(* PLC project Generated.project, CODESYS CODESYS V3.5 SP19 Patch 1 *)
(* stored: creationDateTime 2026-08-31T12:26:56.544484, modificationDateTime 2026-08-31T12:26:56.544484 *)

(* values of E_DiveSearchState: WAIT_PRECONDITIONS: Attente benne ouverte, positions et Kobold au repos; READY_TO_DESCEND: Prêt à assister une demande de descente; SEARCHING_IMMERSION: Descending : attente front 0->1 dans fenêtre eau; SEARCHING_BOTTOM: Immersion validée : attente front 1->0 au fond; BOTTOM_CONFIRMED: Fond validé ; extraction peut être demandée; ERROR_HOLD: Séquence invalide, descente assistée interdite *)

{attribute 'qualified_only'}
{attribute 'strict'}
TYPE E_DiveSearchState : (WAIT_PRECONDITIONS := 0, READY_TO_DESCEND := 1, SEARCHING_IMMERSION := 2, SEARCHING_BOTTOM := 3, BOTTOM_CONFIRMED := 4, ERROR_HOLD := 5);
END_TYPE

(* ======================================================================= 🧩 ST_Fault — Brique socle défaut (2 vues : live + latchée) ─────────────────────────────────────────────────────────────── 🎯 Rôle : porter l'état défaut d'un composant, applicable dans TOUS les cas (acquittable ou non), sans brique warning séparée. • Vue LIVE (Error / ErrorId) : suit la cause, retombe seule à 0. • Vue LATCHÉE (Latched / LatchedId): mémorisée au défaut, reste jusqu'au front Reset. Le choix acquittable / non-acquittable se fait PAR CAUSE (ST_FaultCause.Latching), jamais par bloc. 🔒 Sécurité : interlock TOUJOURS sur la cause brute (Error / ErrorId), jamais sur l'acquittement. Reset TOUJOURS effectif, jamais conditionné (std §9). 🧬 Composition : brique de base réutilisable — sortie de FB, struct métier, GVL. Texte IHM NON stocké ici : dérivé côté IHM depuis LatchedId / ErrorId. 📄 Doc : DOC/STDS/CODE_QUALITY_STANDARDS.md §2quinquies / §9 ======================================================================= *)
TYPE ST_Fault : STRUCT
  Error : BOOL;  (* <-- [DIAG] vue LIVE : au moins une cause présente maintenant *)
  ErrorId : WORD;  (* <-- [DIAG] bitfield des causes présentes maintenant (0 si aucune) *)
  Latched : BOOL;  (* <-- [DIAG] vue LATCHÉE : défaut non acquitté, reste jusqu'au front Reset *)
  LatchedId : WORD;  (* <-- [DIAG] ErrorId figé à l'apparition du défaut, effacé au Reset *)
END_STRUCT;
END_TYPE

(* ======================================================================= 🧩 ST_FaultCause — Cause élémentaire alimentant ST_Fault (socle FB_FaultCore) ─────────────────────────────────────────────────────────────── 🎯 Rôle : une cause exprimée EN CLAIR (BOOL + libellé), sans bitfield ni masque. Le FB métier remplit une liste (ARRAY[0..15] OF ST_FaultCause) ; le socle FB_FaultCore en déduit ST_Fault (vue live + vue latchée). 🔒 Sécurité : interlock TOUJOURS sur Active (cause brute), jamais sur le latch. Latching = TRUE → la cause ARME la vue latchée (défaut à acquitter). Latching = FALSE → la cause n'alimente que la vue live (retombe seule). Fail-safe : une cause laissée à Latching=FALSE reste visible en live — pour la rendre acquittable, il faut le déclarer explicitement. 📄 Doc : DOC/STDS/CODE_QUALITY_STANDARDS.md §2quinquies / §9 ======================================================================= *)
TYPE ST_FaultCause : STRUCT
  Active : BOOL;  (* 1 = cause présente maintenant (interlock sur cette valeur) *)
  Latching : BOOL;  (* 1 = cause à acquitter (arme Latched) ; 0 = live seulement *)
  Texte : STRING;  (* libellé prêt IHM (non stocké dans ST_Fault, dérivé côté IHM) *)
END_STRUCT;
END_TYPE

(* ======================================================================= 🧩 ST_Lifecycle — Brique socle cycle d'exécution ─────────────────────────────────────────────────────────────── 🎯 Rôle : porter l'avancement d'une action à cycle (organe, séquenceur). Optionnelle : un FB purement synchrone (conditionneur, filtre, joystick) ne la porte pas. 🧬 Composition : brique de base réutilisable, composée avec ST_Fault. 📄 Doc : DOC/STDS/CODE_QUALITY_STANDARDS.md §2quinquies ======================================================================= *)
TYPE ST_Lifecycle : STRUCT
  Busy : BOOL;  (* <-- [STAT] 1 = action en cours *)
  Done : BOOL;  (* <-- [STAT] 1 = action terminée avec succès *)
END_STRUCT;
END_TYPE

(* ======================================================================= ST_fbDiveSearch_Inputs - Bus d'entree du cycle FB_DiveSearch ======================================================================= *)
TYPE ST_fbDiveSearch_Inputs : STRUCT
  PowerContactorEngaged : BOOL;  (* === AUTORISATIONS & COMMANDE === Chaine de puissance engagee *)
  Mode : E_Mode;  (* Mode arbitre courant *)
  MotionRequestActive : BOOL;  (* Demande de mouvement couplee *)
  MotionDirection : INT;  (* Sens demande (-1 = descente) *)
  BucketIsOpen : BOOL;  (* === CAPTEURS & MESURES === Benne ouverte confirmee *)
  KoboldImmersed : BOOL;  (* Kobold immerge *)
  M1Position_M : REAL;  (* Position cable M1 (m) *)
  M2Position_M : REAL;  (* Position cable M2 (m) *)
  PositionsValid : BOOL;  (* Mesures M1/M2 valides *)
  CurrentSpeedStep : INT;  (* Palier reel courant (0..5) *)
  DiveStartMin_M : REAL;  (* === REGLAGES METIER === Position minimale avant descente (m) *)
  ImmersionUpper_M : REAL;  (* Borne haute fenetre immersion (m) *)
  ImmersionLower_M : REAL;  (* Borne basse fenetre immersion (m) *)
  CableLimitAscent_M : REAL;  (* Limite haute exploitation (m) *)
  LimitLegalDepthMin_M : REAL;  (* Limite basse legale (m) *)
  CfgDiveFloorStep : INT;  (* Plancher palier descente (0..5) *)
  CycleTime : TIME;  (* Periode d'execution du cycle *)
  BypassPreconditions : BOOL;  (* Bypass reserve au mode maintenance N2/test *)
  Config : ST_fbDiveSearch_Config;  (* Parametres timeout *)
END_STRUCT;
END_TYPE

(* ======================================================================= ST_fbDiveSearch_Outputs - Bus de sortie du cycle FB_DiveSearch ======================================================================= *)
TYPE ST_fbDiveSearch_Outputs : STRUCT
  StepState : E_DiveSearchState;  (* === ETAT DU CYCLE === Etape courante *)
  StepAtFault : E_DiveSearchState;  (* Etape figee au defaut *)
  DescendPermit : BOOL;  (* === PERMIS & ORDRES ASSISTES === Autorisation de descente assistee *)
  KoboldContactorCmd : BOOL;  (* Commande alimentation Kobold (fail-safe, coupe au front de fond) *)
  BottomTouchConfirmed : BOOL;  (* Fond confirme *)
  MinStepDown : INT;  (* Plancher palier descente *)
  OperatorActionId : WORD;  (* === DIAGNOSTIC OPERATEUR === Identifiant numerique de l'action *)
  OperatorAction : STRING(120);  (* Consigne operateur ASCII *)
END_STRUCT;
END_TYPE

(* values of E_Mode: DISABLE: Mode Désactivé / Veille de sécurité (sorties bloquées); MAINT_N1: Manuel Niveau 1 : Pilotage unitaire avec toutes sécurités actives; MAINT_N2: Manuel Niveau 2 : Pilotage dégradé (droits étendus + bypasses autorisés); SEMI_AUTO: Mode Semi-Automatique (séquenceur automatique) *)

{attribute 'qualified_only'}
{attribute 'strict'}
TYPE E_Mode : (DISABLE := 0, MAINT_N1 := 1, MAINT_N2 := 2, SEMI_AUTO := 3);
END_TYPE

(* ======================================================================= ST_fbDiveSearch_Config - Reglages du cycle de recherche du fond ======================================================================= *)
TYPE ST_fbDiveSearch_Config : STRUCT
  DiveSpeedMin_Mps : REAL := 0.15;  (* Vitesse minimale de calcul du timeout (m/s) *)
  TimeoutMarginFactor : REAL := 1.5;  (* Marge appliquee au temps theorique *)
  TimeoutMinCourse_M : REAL := 1;  (* Course minimale prise en compte (m) *)
  TimeoutMaxCourse_M : REAL := 200;  (* Course maximale prise en compte (m) *)
  SecToMs : REAL := 1000;  (* Conversion secondes vers millisecondes *)
END_STRUCT;
END_TYPE

(* ======================================================================= FB_DiveSearch - Assistance plongee et recherche du fond Kobold Role : qualifier l'immersion et autoriser la descente assistee. Interface : contrat standard + bus Inputs/Outputs. Documentation : DOC/AF/AF_Partie-04_Mode_SemiAuto_Sequenceur_v2.3.md ======================================================================= *)
FUNCTION_BLOCK FB_DiveSearch
  VAR_INPUT
    Enable : BOOL;  (* === CONTRAT STANDARD === --> [CMD] Autorisation generale du FB *)
    Reset : BOOL;  (* --> [CMD] Acquittement defaut sur front *)
    Inputs : ST_fbDiveSearch_Inputs;  (* === BUS FONCTIONNEL === --> [BUS] Commande, capteurs et reglages *)
  END_VAR
  VAR_OUTPUT
    Ready : BOOL;  (* === STATUT IEC === <-- [STAT] FB pret a fonctionner *)
    Fault : ST_Fault;  (* <-- [DIAG] Defaut live et latche *)
    Lifecycle : ST_Lifecycle;  (* <-- [STAT] Cycle en cours / termine *)
    Outputs : ST_fbDiveSearch_Outputs;  (* === BUS FONCTIONNEL === <-- [BUS] Etat, permis et diagnostic *)
  END_VAR
  VAR
    ResetEdge : R_TRIG;  (* === SOUS-INSTANCES & FRONTS === . [LOC] Front Reset *)
    ErrorEdge : R_TRIG;  (* . [LOC] Apparition d'un defaut *)
    KoboldRiseEdge : R_TRIG;  (* . [LOC] Entree dans l'eau *)
    KoboldFallEdge : F_TRIG;  (* . [LOC] Sortie de l'eau / fond *)
    instFault : FB_FaultCore;  (* * [INST] Socle defaut transverse *)
    instCauses : ARRAY[0..15] OF ST_FaultCause;  (* . [LOC] Causes nommees *)
    ImmersionCourse_M : REAL;  (* === CALCULS DE GARDE === . [LOC] Course maximale vers immersion (m) *)
    BottomCourse_M : REAL;  (* . [LOC] Course maximale vers fond (m) *)
    CalculatedImmersionTimeout : TIME;  (* . [LOC] Timeout immersion calcule *)
    CalculatedBottomTimeout : TIME;  (* . [LOC] Timeout fond calcule *)
    EffectiveDiveSpeedMin_Mps : REAL;  (* . [LOC] Vitesse minimale appliquee (m/s) *)
    EffectiveTimeoutMargin : REAL;  (* . [LOC] Marge appliquee au calcul *)
    EffectiveTimeoutMinCourse_M : REAL;  (* . [LOC] Plancher de course applique (m) *)
    EffectiveTimeoutMaxCourse_M : REAL;  (* . [LOC] Plafond de course applique (m) *)
    EffectiveSecToMs : REAL;  (* . [LOC] Conversion secondes/millisecondes *)
    ImmersionTimerAcc : TIME := TIME#0ms;  (* === MEMORISATIONS & TEMPORISATIONS === . [LOC] Temps effectif de recherche immersion *)
    BottomTimerAcc : TIME := TIME#0ms;  (* . [LOC] Temps effectif de recherche fond *)
    PrevState : E_DiveSearchState;  (* . [LOC] Etat du scan precedent *)
    ImmersionConfirmed : BOOL;  (* . [LOC] Immersion validee *)
    StepAtFaultCaptured : BOOL;  (* . [LOC] Etape de defaut deja figee *)
    ErrorCausePresent : BOOL;  (* === CAUSES INTERNES === . [LOC] Parametrage invalide *)
    SeqErrorFault : BOOL;  (* . [LOC] Incoherence de sequence *)
    Palier5ForbiddenFault : BOOL;  (* . [LOC] Palier 5 interdit sous Kobold *)
    TimeoutImmersionFault : BOOL;  (* . [LOC] Timeout recherche immersion *)
    TimeoutBottomFault : BOOL;  (* . [LOC] Timeout recherche fond *)
    DescentActive : BOOL;  (* . [LOC] Descending demandee et autorisee *)
  END_VAR

            

{region "§1 Fronts, calculs et causes"}
ResetEdge(CLK := Reset);
KoboldRiseEdge(CLK := Inputs.KoboldImmersed);
KoboldFallEdge(CLK := Inputs.KoboldImmersed);

// Les valeurs par defaut du DUT couvrent l'appel sans configuration explicite.
// Le repli runtime protege aussi un appel avec une structure entierement nulle.
EffectiveDiveSpeedMin_Mps := Inputs.Config.DiveSpeedMin_Mps;
IF EffectiveDiveSpeedMin_Mps <= 0.0 THEN EffectiveDiveSpeedMin_Mps := 0.15; END_IF;
EffectiveTimeoutMargin := Inputs.Config.TimeoutMarginFactor;
IF EffectiveTimeoutMargin <= 0.0 THEN EffectiveTimeoutMargin := 1.5; END_IF;
EffectiveTimeoutMinCourse_M := Inputs.Config.TimeoutMinCourse_M;
IF EffectiveTimeoutMinCourse_M <= 0.0 THEN EffectiveTimeoutMinCourse_M := 1.0; END_IF;
EffectiveTimeoutMaxCourse_M := Inputs.Config.TimeoutMaxCourse_M;
IF EffectiveTimeoutMaxCourse_M < EffectiveTimeoutMinCourse_M THEN EffectiveTimeoutMaxCourse_M := 200.0; END_IF;
EffectiveSecToMs := Inputs.Config.SecToMs;
IF EffectiveSecToMs <= 0.0 THEN EffectiveSecToMs := 1000.0; END_IF;

ErrorCausePresent := (Inputs.CycleTime <= T#0ms)
                 OR (NOT Inputs.BypassPreconditions AND (
                       (Inputs.DiveStartMin_M < Inputs.ImmersionUpper_M)
                    OR (Inputs.ImmersionUpper_M <= Inputs.ImmersionLower_M)
                    OR (Inputs.ImmersionLower_M <= Inputs.LimitLegalDepthMin_M)
                    OR (Inputs.CableLimitAscent_M <= Inputs.ImmersionLower_M)));

ImmersionCourse_M := LIMIT(EffectiveTimeoutMinCourse_M,
                           Inputs.CableLimitAscent_M - Inputs.ImmersionLower_M,
                           EffectiveTimeoutMaxCourse_M);
BottomCourse_M := LIMIT(EffectiveTimeoutMinCourse_M,
                        Inputs.ImmersionLower_M - Inputs.LimitLegalDepthMin_M,
                        EffectiveTimeoutMaxCourse_M);
CalculatedImmersionTimeout := UDINT_TO_TIME(REAL_TO_UDINT(
    ImmersionCourse_M / EffectiveDiveSpeedMin_Mps * EffectiveTimeoutMargin * EffectiveSecToMs));
CalculatedBottomTimeout := UDINT_TO_TIME(REAL_TO_UDINT(
    BottomCourse_M / EffectiveDiveSpeedMin_Mps * EffectiveTimeoutMargin * EffectiveSecToMs));

IF (Outputs.StepState = E_DiveSearchState.SEARCHING_IMMERSION)
   AND Inputs.MotionRequestActive AND (Inputs.MotionDirection = -1) THEN
    ImmersionTimerAcc := ImmersionTimerAcc + Inputs.CycleTime;
    IF ImmersionTimerAcc >= CalculatedImmersionTimeout THEN TimeoutImmersionFault := TRUE; END_IF;
END_IF;

IF (Outputs.StepState = E_DiveSearchState.SEARCHING_BOTTOM)
   AND Inputs.MotionRequestActive AND (Inputs.MotionDirection = -1) THEN
    BottomTimerAcc := BottomTimerAcc + Inputs.CycleTime;
    IF BottomTimerAcc >= CalculatedBottomTimeout THEN TimeoutBottomFault := TRUE; END_IF;
END_IF;

IF ResetEdge.Q AND NOT ErrorCausePresent AND NOT Inputs.KoboldImmersed
   AND NOT Inputs.MotionRequestActive AND NOT (Inputs.CurrentSpeedStep > 4) THEN
    SeqErrorFault := FALSE;
    Palier5ForbiddenFault := FALSE;
    TimeoutImmersionFault := FALSE;
    TimeoutBottomFault := FALSE;
    ImmersionTimerAcc := T#0ms;
    BottomTimerAcc := T#0ms;
    ImmersionConfirmed := FALSE;
    Outputs.BottomTouchConfirmed := FALSE;
    Outputs.StepAtFault := E_DiveSearchState.WAIT_PRECONDITIONS;
    StepAtFaultCaptured := FALSE;
    Outputs.StepState := E_DiveSearchState.WAIT_PRECONDITIONS;
END_IF;

instCauses[0].Active := SeqErrorFault;
instCauses[0].Latching := TRUE;
instCauses[0].Texte := 'Incoherence sequence immersion Kobold';
instCauses[1].Active := ErrorCausePresent;
instCauses[1].Latching := TRUE;
instCauses[1].Texte := 'Parametrage invalide des seuils de plongee';
instCauses[2].Active := Palier5ForbiddenFault;
instCauses[2].Latching := TRUE;
instCauses[2].Texte := 'Palier 5 interdit pendant la mesure Kobold';
instCauses[3].Active := TimeoutImmersionFault;
instCauses[3].Latching := TRUE;
instCauses[3].Texte := 'Timeout recherche immersion Kobold';
instCauses[4].Active := TimeoutBottomFault;
instCauses[4].Latching := TRUE;
instCauses[4].Texte := 'Timeout recherche fond Kobold';

instFault(Enable := Enable, Reset := Reset, Causes := instCauses);
Fault := instFault.Fault;

ErrorEdge(CLK := Fault.Error);
IF ErrorEdge.Q AND NOT StepAtFaultCaptured THEN
    Outputs.StepAtFault := PrevState;
    StepAtFaultCaptured := TRUE;
ELSIF ResetEdge.Q AND NOT ErrorCausePresent AND NOT Inputs.KoboldImmersed
      AND NOT Inputs.MotionRequestActive AND NOT (Inputs.CurrentSpeedStep > 4) THEN
    Outputs.StepAtFault := E_DiveSearchState.WAIT_PRECONDITIONS;
END_IF;
{endregion}

{region "§2 Neutralisation et machine d'etat"}
IF NOT Enable OR NOT Inputs.PowerContactorEngaged THEN
    Ready := FALSE;
    Lifecycle.Busy := FALSE;
    Lifecycle.Done := FALSE;
    Outputs.DescendPermit := FALSE;
    Outputs.KoboldContactorCmd := FALSE;
    Outputs.BottomTouchConfirmed := FALSE;
    Outputs.StepState := E_DiveSearchState.WAIT_PRECONDITIONS;
    Outputs.OperatorActionId := 0;
    Outputs.OperatorAction := '';
    ImmersionConfirmed := FALSE;
    ImmersionTimerAcc := T#0ms;
    BottomTimerAcc := T#0ms;
    Outputs.MinStepDown := 0;
    PrevState := E_DiveSearchState.WAIT_PRECONDITIONS;
    RETURN;
END_IF;

Ready := Enable AND NOT Fault.Latched;
Outputs.DescendPermit := FALSE;
Outputs.KoboldContactorCmd := FALSE;
Lifecycle.Busy := FALSE;
Lifecycle.Done := FALSE;
Outputs.OperatorActionId := 0;
Outputs.OperatorAction := '';

DescentActive := Inputs.MotionRequestActive AND (Inputs.MotionDirection = -1)
              AND ((Inputs.Mode = E_Mode.MAINT_N1) OR (Inputs.Mode = E_Mode.MAINT_N2))
              AND NOT (Inputs.CurrentSpeedStep > 4)
              AND NOT SeqErrorFault;

IF Fault.Error OR Fault.Latched THEN
    Outputs.StepState := E_DiveSearchState.ERROR_HOLD;
    Outputs.KoboldContactorCmd := FALSE;
    Outputs.OperatorActionId := 16#0180;
    Outputs.OperatorAction := 'Verifier les conditions puis rearmer avant une nouvelle plongee.';
ELSE
    CASE Outputs.StepState OF
        E_DiveSearchState.WAIT_PRECONDITIONS:
            IF NOT Inputs.BypassPreconditions
               AND (NOT Inputs.BucketIsOpen OR NOT Inputs.PositionsValid OR Inputs.KoboldImmersed
                    OR (Inputs.M1Position_M < Inputs.DiveStartMin_M)
                    OR (Inputs.M2Position_M < Inputs.DiveStartMin_M)) THEN
                Outputs.OperatorActionId := 16#0100;
                Outputs.OperatorAction := 'Verifier benne ouverte, positions et Kobold au repos.';
            ELSE
                Outputs.StepState := E_DiveSearchState.READY_TO_DESCEND;
            END_IF;

        E_DiveSearchState.READY_TO_DESCEND:
            Ready := TRUE;
            Outputs.OperatorActionId := 16#0101;
            Outputs.OperatorAction := 'Demander une descente pour rechercher le fond.';
            IF Inputs.MotionRequestActive AND (Inputs.MotionDirection = -1) THEN
                ImmersionTimerAcc := T#0ms;
                Outputs.StepState := E_DiveSearchState.SEARCHING_IMMERSION;
            END_IF;

        E_DiveSearchState.SEARCHING_IMMERSION:
            Lifecycle.Busy := TRUE;
            Outputs.DescendPermit := DescentActive;
            Outputs.KoboldContactorCmd := DescentActive;
            Outputs.OperatorActionId := 16#0102;
            Outputs.OperatorAction := 'Maintenir la descente : recherche immersion Kobold.';
            IF Inputs.CurrentSpeedStep > 4 THEN
                IF NOT StepAtFaultCaptured THEN
                    Outputs.StepAtFault := Outputs.StepState;
                    StepAtFaultCaptured := TRUE;
                END_IF;
                Palier5ForbiddenFault := TRUE;
            END_IF;
            IF KoboldRiseEdge.Q THEN
                IF (Inputs.M1Position_M <= Inputs.ImmersionUpper_M)
                   AND (Inputs.M1Position_M >= Inputs.ImmersionLower_M)
                   AND (Inputs.M2Position_M <= Inputs.ImmersionUpper_M)
                   AND (Inputs.M2Position_M >= Inputs.ImmersionLower_M) THEN
                    ImmersionConfirmed := TRUE;
                    BottomTimerAcc := T#0ms;
                    Outputs.StepState := E_DiveSearchState.SEARCHING_BOTTOM;
                ELSE
                    IF NOT StepAtFaultCaptured THEN
                        Outputs.StepAtFault := Outputs.StepState;
                        StepAtFaultCaptured := TRUE;
                    END_IF;
                    SeqErrorFault := TRUE;
                END_IF;
            ELSIF (Inputs.M1Position_M < Inputs.ImmersionLower_M)
               OR (Inputs.M2Position_M < Inputs.ImmersionLower_M) THEN
                IF NOT StepAtFaultCaptured THEN
                    Outputs.StepAtFault := Outputs.StepState;
                    StepAtFaultCaptured := TRUE;
                END_IF;
                SeqErrorFault := TRUE;
            END_IF;

        E_DiveSearchState.SEARCHING_BOTTOM:
            Lifecycle.Busy := TRUE;
            Outputs.DescendPermit := DescentActive;
            Outputs.KoboldContactorCmd := DescentActive;
            Outputs.OperatorActionId := 16#0103;
            Outputs.OperatorAction := 'Maintenir la descente : immersion validee, recherche du fond.';
            IF Inputs.CurrentSpeedStep > 4 THEN
                IF NOT StepAtFaultCaptured THEN
                    Outputs.StepAtFault := Outputs.StepState;
                    StepAtFaultCaptured := TRUE;
                END_IF;
                Palier5ForbiddenFault := TRUE;
            END_IF;
            IF KoboldFallEdge.Q AND ImmersionConfirmed THEN
                Outputs.BottomTouchConfirmed := TRUE;
                ImmersionConfirmed := FALSE;
                Outputs.KoboldContactorCmd := FALSE;
                Outputs.StepState := E_DiveSearchState.BOTTOM_CONFIRMED;
            END_IF;

        E_DiveSearchState.BOTTOM_CONFIRMED:
            Lifecycle.Done := TRUE;
            Outputs.KoboldContactorCmd := FALSE;
            Outputs.OperatorActionId := 16#0104;
            Outputs.OperatorAction := 'Fond detecte : demander la fermeture ou extraction.';

        E_DiveSearchState.ERROR_HOLD:
            Outputs.KoboldContactorCmd := FALSE;
    END_CASE;
END_IF;

IF DescentActive AND ((Outputs.StepState = E_DiveSearchState.SEARCHING_IMMERSION)
                   OR (Outputs.StepState = E_DiveSearchState.SEARCHING_BOTTOM)) THEN
    Outputs.MinStepDown := LIMIT(0, Inputs.CfgDiveFloorStep, 5);
ELSE
    Outputs.MinStepDown := 0;
END_IF;

PrevState := Outputs.StepState;
{endregion}

          
END_FUNCTION_BLOCK

(* ======================================================================= 🧩 FB_FaultCore — Socle de remplissage de ST_Fault (vue live + vue latchée) ─────────────────────────────────────────────────────────────── 🎯 Rôle : à partir d'une LISTE de causes en clair (ARRAY[0..15] OF ST_FaultCause), produire la brique ST_Fault : • Error / ErrorId : vue LIVE, suit les causes Active, retombe seule. • Latched / LatchedId: vue LATCHÉE, chaque bit figé à l'apparition d'une cause `Active AND Latching`, conservé jusqu'au front Reset. 🔒 Sécurité : - interlock TOUJOURS sur `Causes[i].Active` (cause brute), jamais sur le latch. - Reset TOUJOURS effectif, jamais conditionné (std §9) — agit même Enable=FALSE. - Latching=FALSE → cause visible en LIVE seulement (fail-safe : reste visible). - un défaut laté non acquitté reste publié même FB désactivé (pas d'effacement silencieux sur bascule Enable OFF→ON sans Reset). - une cause à acquitter réapparue re-arme son bit (ré-alarme). 🧬 Un seul socle, réutilisé par tout FB `standard` qui expose un ST_Fault. Pas de State, pas de Warning, pas de texte — hors périmètre de ce socle. 📄 Doc : DOC/STDS/CODE_QUALITY_STANDARDS.md §2quinquies / §9 ======================================================================= *)
FUNCTION_BLOCK FB_FaultCore
  VAR_INPUT
    Enable : BOOL;  (* --> [CMD] Autorisation générale du FB porteur *)
    Reset : BOOL;  (* --> [CMD] Front d'acquittement (jamais conditionné, §9) *)
    Causes : ARRAY[0..15] OF ST_FaultCause;  (* --> [CMD] Liste des causes en clair (Active / Latching / Texte) *)
  END_VAR
  VAR_OUTPUT
    Ready : BOOL;  (* <-- [STAT] FB porteur autorisé (= Enable) *)
    Fault : ST_Fault;  (* <-- [DIAG] Brique défaut (mappée 1:1 sur la sortie du FB porteur) *)
  END_VAR
  VAR
    ResetEdge : R_TRIG;  (* . [LOC] Front montant Reset *)
    Latch : ARRAY[0..15] OF BOOL;  (* . [LOC] Bit laté par cause, jusqu'au Reset *)
    i : INT;  (* . [LOC] Index de parcours de la liste *)
  END_VAR

            

{region "§1 Reset (front, toujours effectif)"}
// Front Reset : efface tous les latches. Jamais conditionné, agit même Enable=FALSE (§9).
Ready := Enable;
ResetEdge(CLK := Reset);
IF ResetEdge.Q THEN
    FOR i := 0 TO 15 DO Latch[i] := FALSE; END_FOR;
END_IF;
{endregion}

{region "§2 Vue LIVE — Error / ErrorId"}
// Bitfield des causes présentes MAINTENANT. Retombe seule à 0 quand les causes disparaissent.
// Non évaluée si Enable=FALSE (pas de lecture de cause hors autorisation).
Fault.ErrorId := 0;
IF Enable THEN
    FOR i := 0 TO 15 DO
        IF Causes[i].Active THEN
            Fault.ErrorId := Fault.ErrorId OR SHL(WORD#1, INT_TO_DWORD(i));
        END_IF;
    END_FOR;
END_IF;
Fault.Error := (Fault.ErrorId <> 0);
{endregion}

{region "§3 Armement des latches (causes à acquitter)"}
// Une cause Active ET Latching arme son bit ; le bit reste jusqu'au front Reset (§1),
// même si la cause disparaît. Réapparition => ré-armement (ré-alarme).
IF Enable THEN
    FOR i := 0 TO 15 DO
        IF Causes[i].Active AND Causes[i].Latching THEN
            Latch[i] := TRUE;
        END_IF;
    END_FOR;
END_IF;
{endregion}

{region "§4 Vue LATCHÉE — Latched / LatchedId"}
// Toujours publiée, y compris Enable=FALSE : un défaut non acquitté reste visible.
Fault.LatchedId := 0;
FOR i := 0 TO 15 DO
    IF Latch[i] THEN
        Fault.LatchedId := Fault.LatchedId OR SHL(WORD#1, INT_TO_DWORD(i));
    END_IF;
END_FOR;
Fault.Latched := (Fault.LatchedId <> 0);
{endregion}

          
END_FUNCTION_BLOCK
